FUNCTION ASSEMBLE_LWORD_FROM_QUARTERS (* this Function combines the 31 QUARTER BYTES to a LWORD *)
  (* Standard: 61499-1; Description: Copyright (c) 2024 HR Agrartechnik GmbH This program and the accompanying materials are made available under the terms of the Eclipse Public License 2.0 which is available at https://www.eclipse.org/legal/epl-2.0/ SPDX-License-Identifier: EPL-2.0 *)
  (* Version 3.0.1, 2026-09-29, Martin Jobst, fix ST package declaration *)
  (* Version 3.0, 2025-04-14, Patrick Aigner, changed package *)
  (* Version 1.1, 2024-07-28, Moritz Ortmeier, HR Agrartechnik, rename Function and change Input/Output Variables *)
  (* Version 1.0, 2024-02-22, Franz Höpfinger, HR Agrartechnik, initial Implementation *)
  PACKAGE eclipse4diac::utils::assembling;
  IMPORT eclipse4diac::utils::const::quarterconst;
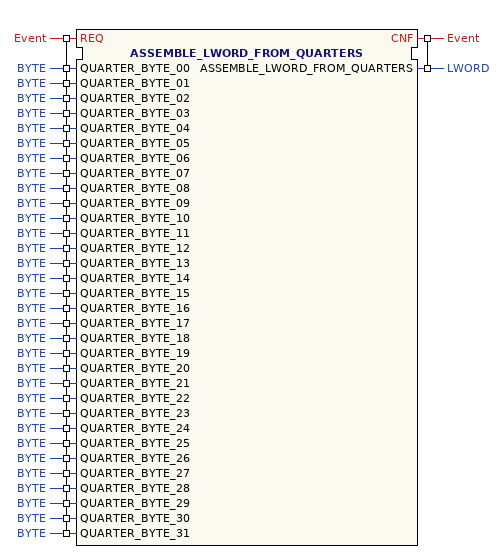
  EVENT_INPUT
    REQ WITH QUARTER_BYTE_00, QUARTER_BYTE_01, QUARTER_BYTE_02, QUARTER_BYTE_03, QUARTER_BYTE_04, QUARTER_BYTE_05, QUARTER_BYTE_06, QUARTER_BYTE_07, QUARTER_BYTE_08, QUARTER_BYTE_09, QUARTER_BYTE_10, QUARTER_BYTE_11, QUARTER_BYTE_12, QUARTER_BYTE_13, QUARTER_BYTE_14, QUARTER_BYTE_15, QUARTER_BYTE_16, QUARTER_BYTE_17, QUARTER_BYTE_18, QUARTER_BYTE_19, QUARTER_BYTE_20, QUARTER_BYTE_21, QUARTER_BYTE_22, QUARTER_BYTE_23, QUARTER_BYTE_24, QUARTER_BYTE_25, QUARTER_BYTE_26, QUARTER_BYTE_27, QUARTER_BYTE_28, QUARTER_BYTE_29, QUARTER_BYTE_30, QUARTER_BYTE_31;
  END_EVENT
  EVENT_OUTPUT
    CNF WITH ASSEMBLE_LWORD_FROM_QUARTERS;
  END_EVENT
  VAR_INPUT
    QUARTER_BYTE_00 : BYTE;
    QUARTER_BYTE_01 : BYTE;
    QUARTER_BYTE_02 : BYTE;
    QUARTER_BYTE_03 : BYTE;
    QUARTER_BYTE_04 : BYTE;
    QUARTER_BYTE_05 : BYTE;
    QUARTER_BYTE_06 : BYTE;
    QUARTER_BYTE_07 : BYTE;
    QUARTER_BYTE_08 : BYTE;
    QUARTER_BYTE_09 : BYTE;
    QUARTER_BYTE_10 : BYTE;
    QUARTER_BYTE_11 : BYTE;
    QUARTER_BYTE_12 : BYTE;
    QUARTER_BYTE_13 : BYTE;
    QUARTER_BYTE_14 : BYTE;
    QUARTER_BYTE_15 : BYTE;
    QUARTER_BYTE_16 : BYTE;
    QUARTER_BYTE_17 : BYTE;
    QUARTER_BYTE_18 : BYTE;
    QUARTER_BYTE_19 : BYTE;
    QUARTER_BYTE_20 : BYTE;
    QUARTER_BYTE_21 : BYTE;
    QUARTER_BYTE_22 : BYTE;
    QUARTER_BYTE_23 : BYTE;
    QUARTER_BYTE_24 : BYTE;
    QUARTER_BYTE_25 : BYTE;
    QUARTER_BYTE_26 : BYTE;
    QUARTER_BYTE_27 : BYTE;
    QUARTER_BYTE_28 : BYTE;
    QUARTER_BYTE_29 : BYTE;
    QUARTER_BYTE_30 : BYTE;
    QUARTER_BYTE_31 : BYTE;
  END_VAR
  VAR_OUTPUT
    ASSEMBLE_LWORD_FROM_QUARTERS : LWORD;
  END_VAR
  BODY IN ST:
PACKAGE eclipse4diac::utils::assembling;

IMPORT eclipse4diac::utils::const::quarterconst;

(* this Function combines the 31 QUARTER BYTES to a LWORD *)
FUNCTION ASSEMBLE_LWORD_FROM_QUARTERS : LWORD

VAR_INPUT
	QUARTER_BYTE_00 : BYTE;
	QUARTER_BYTE_01 : BYTE;
	QUARTER_BYTE_02 : BYTE;
	QUARTER_BYTE_03 : BYTE;
	QUARTER_BYTE_04 : BYTE;
	QUARTER_BYTE_05 : BYTE;
	QUARTER_BYTE_06 : BYTE;
	QUARTER_BYTE_07 : BYTE;
	QUARTER_BYTE_08 : BYTE;
	QUARTER_BYTE_09 : BYTE;
	QUARTER_BYTE_10 : BYTE;
	QUARTER_BYTE_11 : BYTE;
	QUARTER_BYTE_12 : BYTE;
	QUARTER_BYTE_13 : BYTE;
	QUARTER_BYTE_14 : BYTE;
	QUARTER_BYTE_15 : BYTE;
	QUARTER_BYTE_16 : BYTE;
	QUARTER_BYTE_17 : BYTE;
	QUARTER_BYTE_18 : BYTE;
	QUARTER_BYTE_19 : BYTE;
	QUARTER_BYTE_20 : BYTE;
	QUARTER_BYTE_21 : BYTE;
	QUARTER_BYTE_22 : BYTE;
	QUARTER_BYTE_23 : BYTE;
	QUARTER_BYTE_24 : BYTE;
	QUARTER_BYTE_25 : BYTE;
	QUARTER_BYTE_26 : BYTE;
	QUARTER_BYTE_27 : BYTE;
	QUARTER_BYTE_28 : BYTE;
	QUARTER_BYTE_29 : BYTE;
	QUARTER_BYTE_30 : BYTE;
	QUARTER_BYTE_31 : BYTE;
END_VAR

ASSEMBLE_LWORD_FROM_QUARTERS := quarterconst::LWORD_QUARTER_ZZ;
ASSEMBLE_LWORD_FROM_QUARTERS := ASSEMBLE_LWORD_FROM_QUARTERS
	OR SHL(BYTE_TO_LWORD(QUARTER_BYTE_31), quarterconst::SHIFT_QUARTER_31);
ASSEMBLE_LWORD_FROM_QUARTERS := ASSEMBLE_LWORD_FROM_QUARTERS
	OR SHL(BYTE_TO_LWORD(QUARTER_BYTE_30), quarterconst::SHIFT_QUARTER_30);
ASSEMBLE_LWORD_FROM_QUARTERS := ASSEMBLE_LWORD_FROM_QUARTERS
	OR SHL(BYTE_TO_LWORD(QUARTER_BYTE_29), quarterconst::SHIFT_QUARTER_29);
ASSEMBLE_LWORD_FROM_QUARTERS := ASSEMBLE_LWORD_FROM_QUARTERS
	OR SHL(BYTE_TO_LWORD(QUARTER_BYTE_28), quarterconst::SHIFT_QUARTER_28);
ASSEMBLE_LWORD_FROM_QUARTERS := ASSEMBLE_LWORD_FROM_QUARTERS
	OR SHL(BYTE_TO_LWORD(QUARTER_BYTE_27), quarterconst::SHIFT_QUARTER_27);
ASSEMBLE_LWORD_FROM_QUARTERS := ASSEMBLE_LWORD_FROM_QUARTERS
	OR SHL(BYTE_TO_LWORD(QUARTER_BYTE_26), quarterconst::SHIFT_QUARTER_26);
ASSEMBLE_LWORD_FROM_QUARTERS := ASSEMBLE_LWORD_FROM_QUARTERS
	OR SHL(BYTE_TO_LWORD(QUARTER_BYTE_25), quarterconst::SHIFT_QUARTER_25);
ASSEMBLE_LWORD_FROM_QUARTERS := ASSEMBLE_LWORD_FROM_QUARTERS
	OR SHL(BYTE_TO_LWORD(QUARTER_BYTE_24), quarterconst::SHIFT_QUARTER_24);
ASSEMBLE_LWORD_FROM_QUARTERS := ASSEMBLE_LWORD_FROM_QUARTERS
	OR SHL(BYTE_TO_LWORD(QUARTER_BYTE_23), quarterconst::SHIFT_QUARTER_23);
ASSEMBLE_LWORD_FROM_QUARTERS := ASSEMBLE_LWORD_FROM_QUARTERS
	OR SHL(BYTE_TO_LWORD(QUARTER_BYTE_22), quarterconst::SHIFT_QUARTER_22);
ASSEMBLE_LWORD_FROM_QUARTERS := ASSEMBLE_LWORD_FROM_QUARTERS
	OR SHL(BYTE_TO_LWORD(QUARTER_BYTE_21), quarterconst::SHIFT_QUARTER_21);
ASSEMBLE_LWORD_FROM_QUARTERS := ASSEMBLE_LWORD_FROM_QUARTERS
	OR SHL(BYTE_TO_LWORD(QUARTER_BYTE_20), quarterconst::SHIFT_QUARTER_20);
ASSEMBLE_LWORD_FROM_QUARTERS := ASSEMBLE_LWORD_FROM_QUARTERS
	OR SHL(BYTE_TO_LWORD(QUARTER_BYTE_19), quarterconst::SHIFT_QUARTER_19);
ASSEMBLE_LWORD_FROM_QUARTERS := ASSEMBLE_LWORD_FROM_QUARTERS
	OR SHL(BYTE_TO_LWORD(QUARTER_BYTE_18), quarterconst::SHIFT_QUARTER_18);
ASSEMBLE_LWORD_FROM_QUARTERS := ASSEMBLE_LWORD_FROM_QUARTERS
	OR SHL(BYTE_TO_LWORD(QUARTER_BYTE_17), quarterconst::SHIFT_QUARTER_17);
ASSEMBLE_LWORD_FROM_QUARTERS := ASSEMBLE_LWORD_FROM_QUARTERS
	OR SHL(BYTE_TO_LWORD(QUARTER_BYTE_16), quarterconst::SHIFT_QUARTER_16);
ASSEMBLE_LWORD_FROM_QUARTERS := ASSEMBLE_LWORD_FROM_QUARTERS
	OR SHL(BYTE_TO_LWORD(QUARTER_BYTE_15), quarterconst::SHIFT_QUARTER_15);
ASSEMBLE_LWORD_FROM_QUARTERS := ASSEMBLE_LWORD_FROM_QUARTERS
	OR SHL(BYTE_TO_LWORD(QUARTER_BYTE_14), quarterconst::SHIFT_QUARTER_14);
ASSEMBLE_LWORD_FROM_QUARTERS := ASSEMBLE_LWORD_FROM_QUARTERS
	OR SHL(BYTE_TO_LWORD(QUARTER_BYTE_13), quarterconst::SHIFT_QUARTER_13);
ASSEMBLE_LWORD_FROM_QUARTERS := ASSEMBLE_LWORD_FROM_QUARTERS
	OR SHL(BYTE_TO_LWORD(QUARTER_BYTE_12), quarterconst::SHIFT_QUARTER_12);
ASSEMBLE_LWORD_FROM_QUARTERS := ASSEMBLE_LWORD_FROM_QUARTERS
	OR SHL(BYTE_TO_LWORD(QUARTER_BYTE_11), quarterconst::SHIFT_QUARTER_11);
ASSEMBLE_LWORD_FROM_QUARTERS := ASSEMBLE_LWORD_FROM_QUARTERS
	OR SHL(BYTE_TO_LWORD(QUARTER_BYTE_10), quarterconst::SHIFT_QUARTER_10);
ASSEMBLE_LWORD_FROM_QUARTERS := ASSEMBLE_LWORD_FROM_QUARTERS
	OR SHL(BYTE_TO_LWORD(QUARTER_BYTE_09), quarterconst::SHIFT_QUARTER_09);
ASSEMBLE_LWORD_FROM_QUARTERS := ASSEMBLE_LWORD_FROM_QUARTERS
	OR SHL(BYTE_TO_LWORD(QUARTER_BYTE_08), quarterconst::SHIFT_QUARTER_08);
ASSEMBLE_LWORD_FROM_QUARTERS := ASSEMBLE_LWORD_FROM_QUARTERS
	OR SHL(BYTE_TO_LWORD(QUARTER_BYTE_07), quarterconst::SHIFT_QUARTER_07);
ASSEMBLE_LWORD_FROM_QUARTERS := ASSEMBLE_LWORD_FROM_QUARTERS
	OR SHL(BYTE_TO_LWORD(QUARTER_BYTE_06), quarterconst::SHIFT_QUARTER_06);
ASSEMBLE_LWORD_FROM_QUARTERS := ASSEMBLE_LWORD_FROM_QUARTERS
	OR SHL(BYTE_TO_LWORD(QUARTER_BYTE_05), quarterconst::SHIFT_QUARTER_05);
ASSEMBLE_LWORD_FROM_QUARTERS := ASSEMBLE_LWORD_FROM_QUARTERS
	OR SHL(BYTE_TO_LWORD(QUARTER_BYTE_04), quarterconst::SHIFT_QUARTER_04);
ASSEMBLE_LWORD_FROM_QUARTERS := ASSEMBLE_LWORD_FROM_QUARTERS
	OR SHL(BYTE_TO_LWORD(QUARTER_BYTE_03), quarterconst::SHIFT_QUARTER_03);
ASSEMBLE_LWORD_FROM_QUARTERS := ASSEMBLE_LWORD_FROM_QUARTERS
	OR SHL(BYTE_TO_LWORD(QUARTER_BYTE_02), quarterconst::SHIFT_QUARTER_02);
ASSEMBLE_LWORD_FROM_QUARTERS := ASSEMBLE_LWORD_FROM_QUARTERS
	OR SHL(BYTE_TO_LWORD(QUARTER_BYTE_01), quarterconst::SHIFT_QUARTER_01);
ASSEMBLE_LWORD_FROM_QUARTERS := ASSEMBLE_LWORD_FROM_QUARTERS
	OR SHL(BYTE_TO_LWORD(QUARTER_BYTE_00), quarterconst::SHIFT_QUARTER_00);

END_FUNCTION
  END_BODY
END_FUNCTION
